{attribute 'qualified_only'}
{attribute 'strict'}
TYPE eSelectTMCFile :
(
	eDontUseTMCFile	:= 0,
	eUseTMCFile		:= 1
);
END_TYPE

(* stored: Version 1.1.0.1, ProductVersion 3.1.4024.11
   DUT eSelectTMCFile: Id {78fa1bdf-9a33-4286-9227-a41c2841a00a} *)
